PROGRAM POU
VAR
	tVar : TIME := T#5S;
	nRefVar : REFERENCE TO TIME REF= tVar;
END_VAR

nRefVar := T#1S;

END_PROGRAM

(* stored: Version 1.1.0.1, ProductVersion 3.1.4024.12
   POU POU: Id {25bb10e9-007a-4fe5-ae87-87690b6561fa}, SpecialFunc None *)
